// TIA Portal V16 export
// export: Created 2022-11-17T15:49:44.3342436Z, ExportSetting WithDefaults, DisplayName Totally Integrated Automation Portal, DisplayVersion V16 Update 6, DisplayName TIA Portal Version Control Interface, DisplayVersion V16 Update 2, DisplayName TIA Portal Openness, DisplayVersion V16 Update 6, DisplayName SINAMICS Startdrive Advanced, DisplayVersion V16 Update 5, DisplayName SINAMICS Startdrive G130, G150, S120, S150, SINAMICS MV, S210, DisplayVersion V16 Update 5, DisplayName SINAMICS Startdrive G110M, G120, G120C, G120D, G120P, G115D, DisplayVersion V16 Update 5, DisplayName STEP 7 Professional, DisplayVersion V16 Update 6, DisplayName STEP 7 Safety, DisplayVersion V16, DisplayName WinCC Advanced, DisplayVersion V16 Update 6
DATA_BLOCK "DB240_Program10"   // DB240
{ S7_Optimized_Access := 'FALSE' }
AUTHOR : Robopac
VERSION : 0.0
// stored: AutoNumber false, IsOnlyStoredInLoadMemory false, IsWriteProtectedInAS false
   VAR RETAIN
      Program10 { S7_SetPoint := 'True'} : "DatiProgramma";
   END_VAR
BEGIN
   Program10.Wrapping := TRUE;
   Program10.TopLenght := 500;
   Program10.TopRelease := 0;
   Program10.TopDown := 0;
   Program10.Top := 4;
   Program10.PressurePTime := 0;
   Program10.LifterTime := 0;
   Program10.RevOverContrast := 1;
   Program10.RopeEndCycle := 16#02;
   Program10.Spare4 := 16#01;
   Program10.RopeTime := 1500;
   Program10.RevOverClamp := 1;
   Program10.FilmForceFinalRev := 10;
   Program10.FilmPrestretchFinalRev := 100;
   Program10.ArmSpeed := 100;
   Program10.CarriageDown4Top := 500;
   Program10.TopDownTime := 1500;
   Program10.LapsUnderTop := 0;
   Program10.Spare6 := 0;
   Program10.Spare7 := 0;
   Program10.Spare8 := 0;
   Program10.Spare9 := 0;
   Program10.Spare10 := 0;
   Program10.Spare11 := 0;
   Program10.Spare12 := 0;
   Program10.Overlap0_1 := 0;
   Program10.Height1 := 130;
   Program10.Landmark1 := FALSE;
   Program10.Lifter1 := FALSE;
   Program10.SpareBit1H1 := FALSE;
   Program10.Airblower1 := TRUE;
   Program10.NextStep1 := TRUE;
   Program10.PressureP1 := TRUE;
   Program10.SpareByte2H1 := 16#00;
   Program10.Revolution1 := 1;
   Program10.RopeUnit1_1 := 16#01;
   Program10.RopeUnit1_2 := 16#01;
   Program10.FilmForce1 := 5;
   Program10.FilmPrestretch1 := 200;
   Program10.Spare3H1 := 0;
   Program10.Spare49 := 0;
   Program10.Spare50 := 0;
   Program10.Spare51 := 0;
   Program10.Spare52 := 0;
   Program10.Spare53 := 0;
   Program10.Overlap1_2 := 0;
   Program10.Height2 := 50;
   Program10.Landmark2 := FALSE;
   Program10.Lifter2 := FALSE;
   Program10.SpareBit1H2 := FALSE;
   Program10.Airblower2 := TRUE;
   Program10.NextStep2 := TRUE;
   Program10.PressureP2 := TRUE;
   Program10.SpareByte2H2 := 16#00;
   Program10.Revolution2 := 1;
   Program10.RopeUnit2_1 := 16#01;
   Program10.RopeUnit2_2 := 16#01;
   Program10.FilmForce2 := 20;
   Program10.FilmPrestretch2 := 200;
   Program10.Spare3H2 := 0;
   Program10.Spare54 := 0;
   Program10.Spare55 := 0;
   Program10.Spare56 := 0;
   Program10.Spare57 := 0;
   Program10.Spare58 := 0;
   Program10.Overlap2_3 := 100;
   Program10.Height3 := -50;
   Program10.Landmark3 := TRUE;
   Program10.Lifter3 := FALSE;
   Program10.SpareBit1H3 := FALSE;
   Program10.Airblower3 := TRUE;
   Program10.NextStep3 := TRUE;
   Program10.PressureP3 := TRUE;
   Program10.SpareByte2H3 := 16#00;
   Program10.Revolution3 := 2;
   Program10.RopeUnit3_1 := 16#01;
   Program10.RopeUnit3_2 := 16#01;
   Program10.FilmForce3 := 30;
   Program10.FilmPrestretch3 := 200;
   Program10.Spare3H3 := 0;
   Program10.Spare59 := 0;
   Program10.Spare60 := 0;
   Program10.Spare61 := 380;
   Program10.Spare62 := 2800;
   Program10.Spare63 := 0;
   Program10.Overlap3_4 := 100;
   Program10.Height4 := 100;
   Program10.Landmark4 := FALSE;
   Program10.Lifter4 := FALSE;
   Program10.SpareBit1H4 := FALSE;
   Program10.Airblower4 := TRUE;
   Program10.NextStep4 := TRUE;
   Program10.PressureP4 := TRUE;
   Program10.SpareByte2H4 := 16#00;
   Program10.Revolution4 := 3;
   Program10.RopeUnit4_1 := 16#02;
   Program10.RopeUnit4_2 := 16#02;
   Program10.FilmForce4 := 30;
   Program10.FilmPrestretch4 := 200;
   Program10.Spare3H4 := 0;
   Program10.Spare64 := 0;
   Program10.Spare65 := 0;
   Program10.Spare66 := 0;
   Program10.Spare67 := 0;
   Program10.Spare68 := 0;
   Program10.Overlap4_5 := 0;
   Program10.Height5 := 50;
   Program10.Landmark5 := FALSE;
   Program10.Lifter5 := FALSE;
   Program10.SpareBit1H5 := FALSE;
   Program10.Airblower5 := TRUE;
   Program10.NextStep5 := FALSE;
   Program10.PressureP5 := FALSE;
   Program10.SpareByte2H5 := 16#00;
   Program10.Revolution5 := 1;
   Program10.RopeUnit5_1 := 16#01;
   Program10.RopeUnit5_2 := 16#01;
   Program10.FilmForce5 := 30;
   Program10.FilmPrestretch5 := 200;
   Program10.Spare3H5 := 0;
   Program10.Spare69 := 0;
   Program10.Spare70 := 0;
   Program10.Spare71 := 0;
   Program10.Spare72 := 0;
   Program10.Spare73 := 0;
   Program10.Overlap5_6 := 100;
   Program10.Height6 := 50;
   Program10.Landmark6 := FALSE;
   Program10.Lifter6 := FALSE;
   Program10.SpareBit1H6 := FALSE;
   Program10.Airblower6 := TRUE;
   Program10.NextStep6 := FALSE;
   Program10.PressureP6 := FALSE;
   Program10.SpareByte2H6 := 16#00;
   Program10.Revolution6 := 2;
   Program10.RopeUnit6_1 := 16#02;
   Program10.RopeUnit6_2 := 16#01;
   Program10.FilmForce6 := 20;
   Program10.FilmPrestretch6 := 200;
   Program10.Spare3H6 := 0;
   Program10.Spare74 := 0;
   Program10.Spare75 := 0;
   Program10.Spare76 := 0;
   Program10.Spare77 := 0;
   Program10.Spare78 := 0;
   Program10.Overlap6_7 := 0;
   Program10.Height7 := 0;
   Program10.Landmark7 := FALSE;
   Program10.Lifter7 := FALSE;
   Program10.SpareBit1H7 := FALSE;
   Program10.Airblower7 := FALSE;
   Program10.NextStep7 := TRUE;
   Program10.PressureP7 := FALSE;
   Program10.SpareByte2H7 := 16#00;
   Program10.Revolution7 := 1;
   Program10.RopeUnit7_1 := 16#01;
   Program10.RopeUnit7_2 := 16#01;
   Program10.FilmForce7 := 0;
   Program10.FilmPrestretch7 := 100;
   Program10.Spare3H7 := 0;
   Program10.Spare79 := 0;
   Program10.Spare80 := 0;
   Program10.Spare81 := 0;
   Program10.Spare82 := 0;
   Program10.Spare83 := 0;
   Program10.Overlap7_8 := 0;
   Program10.Height8 := 0;
   Program10.Landmark8 := FALSE;
   Program10.Lifter8 := FALSE;
   Program10.SpareBit1H8 := FALSE;
   Program10.Airblower8 := FALSE;
   Program10.NextStep8 := TRUE;
   Program10.PressureP8 := FALSE;
   Program10.SpareByte2H8 := 16#00;
   Program10.Revolution8 := 1;
   Program10.RopeUnit8_1 := 16#01;
   Program10.RopeUnit8_2 := 16#01;
   Program10.FilmForce8 := 0;
   Program10.FilmPrestretch8 := 100;
   Program10.Spare3H8 := 0;
   Program10.Spare84 := 0;
   Program10.Spare85 := 0;
   Program10.Spare86 := 0;
   Program10.Spare87 := 0;
   Program10.Spare88 := 0;
   Program10.Overlap8_9 := 0;
   Program10.Height9 := 0;
   Program10.Landmark9 := FALSE;
   Program10.Lifter9 := FALSE;
   Program10.SpareBit1H9 := FALSE;
   Program10.Airblower9 := FALSE;
   Program10.NextStep9 := TRUE;
   Program10.PressureP9 := FALSE;
   Program10.SpareByte2H9 := 16#00;
   Program10.Revolution9 := 1;
   Program10.RopeUnit9_1 := 16#01;
   Program10.RopeUnit9_2 := 16#01;
   Program10.FilmForce9 := 0;
   Program10.FilmPrestretch9 := 100;
   Program10.Spare3H9 := 0;
   Program10.Spare89 := 0;
   Program10.Spare90 := 0;
   Program10.Spare91 := 0;
   Program10.Spare92 := 0;
   Program10.Spare93 := 0;
   Program10.Overlap9_10 := 0;
   Program10.Height10 := 0;
   Program10.Landmark10 := FALSE;
   Program10.Lifter10 := FALSE;
   Program10.SpareBit1H10 := FALSE;
   Program10.Airblower10 := FALSE;
   Program10.NextStep10 := FALSE;
   Program10.PressureP10 := FALSE;
   Program10.SpareByte2H10 := 16#00;
   Program10.Revolution10 := 1;
   Program10.RopeUnit10_1 := 16#01;
   Program10.RopeUnit10_2 := 16#01;
   Program10.FilmForce10 := 0;
   Program10.FilmPrestretch10 := 100;
   Program10.Spare3H10 := 0;
   Program10.Spare94 := 0;
   Program10.Spare95 := 0;
   Program10.Spare96 := 0;
   Program10.Spare97 := 0;
   Program10.Spare98 := 0;
   Program10.Overlap10_11 := 0;
   Program10.Height11 := 0;
   Program10.Landmark11 := FALSE;
   Program10.Lifter11 := FALSE;
   Program10.SpareBit1H11 := FALSE;
   Program10.Airblower11 := FALSE;
   Program10.NextStep11 := TRUE;
   Program10.PressureP11 := FALSE;
   Program10.SpareByte2H11 := 16#00;
   Program10.Revolution11 := 1;
   Program10.RopeUnit11_1 := 16#01;
   Program10.RopeUnit11_2 := 16#01;
   Program10.FilmForce11 := 0;
   Program10.FilmPrestretch11 := 100;
   Program10.Spare3H11 := 0;
   Program10.Spare99 := 0;
   Program10.Spare100 := 0;
   Program10.Spare101 := 0;
   Program10.Spare102 := 0;
   Program10.Spare103 := 0;
   Program10.Overlap11_12 := 0;
   Program10.Height12 := 0;
   Program10.Landmark12 := FALSE;
   Program10.Lifter12 := FALSE;
   Program10.SpareBit1H12 := FALSE;
   Program10.Airblower12 := FALSE;
   Program10.NextStep12 := FALSE;
   Program10.PressureP12 := FALSE;
   Program10.SpareByte2H12 := 16#00;
   Program10.Revolution12 := 1;
   Program10.RopeUnit12_1 := 16#01;
   Program10.RopeUnit12_2 := 16#01;
   Program10.FilmForce12 := 0;
   Program10.FilmPrestretch12 := 100;
   Program10.Spare3H12 := 0;
   Program10.Spare104 := 0;
   Program10.Spare105 := 0;
   Program10.Spare106 := 0;
   Program10.Spare107 := 0;
   Program10.Spare108 := 0;
END_DATA_BLOCK
